(* IEC 61131-3 sources: AXOpen/src/components.siem.identification/ctrl/src/IdentProfile/AxoIdentificationDataTypes, 3 files *)

(* ---- Axo_IID_CMD_STRUCT.st ---- *)
NAMESPACE AXOpen.Components.Siem.Identification
    {S7.extern=ReadWrite}
    CLASS PUBLIC Axo_IID_CMD_STRUCT
        VAR PUBLIC
            CMD			    :   eAxo_IID_COMMANDS;	                    //Command ID
            ATTRIBUTES	    :   BYTE                    :=  BYTE#16#0;	//Subcommands
            OFFSETBUFFER    :   UINT                    :=  UINT#0;     //Offset for receive buffer
            EPCID_UID	    :   ARRAY[1..62] OF BYTE;
            LEN_DATA	    :   WORD                    :=WORD#16#0;	//Length of data
            ADDR_TAG	    :   DWORD                   :=DWORD#16#0;	//physical address on tag
            CONFIG		    :   BYTE                    :=BYTE#16#0;	//Config Mode for Init
            CHAINED		    :   BOOL                    :=FALSE;		//Chained Bit: 1= chained; 0=unchained
            EXT_UHF		    :   Axo_IID_IN_EXT_UHF;	                    //further Atrributes for extended UHF commands
        END_VAR
    END_CLASS
END_NAMESPACE

(* ---- Axo_IID_HW_CONNECT.st ---- *)
NAMESPACE AXOpen.Components.Siem.Identification
(*
+-----------+-------------------------------------------+------------------------------------------------------+---------------------+
|           |             RF61xR/RF68xR                 |                     RF1xxC/RF360R                    |   RF180C/RF170C/MV  |
| Parameter +----------+----------+----------+----------+----------+----------+----------+----------+----------+----------+----------+
|			|   CH01   |   CH02   |   CH03   |   CH04   |   CH01   |   CH02   |   CH03   |   CH04   |CM_CONFIG |   CH01   |   CH02   |
+===========+==========+==========+==========+==========+==========+==========+==========+==========+==========+==========+==========+
| API       | 16#5B00  | 16#5B00  | 16#5B00  | 16#5B00  | 16#5B00  | 16#5B00  | 16#5B00  | 16#5B00  | 16#5B00  |   16#00  |   16#00  |
+-----------+----------+----------+----------+----------+----------+----------+----------+----------+----------+----------+----------+
| SLOT      |     1    |     1    |     1    |     1    |     2    |     3    |     4    |     5    |     1    |     1    |     1    |
+-----------+----------+----------+----------+----------+----------+----------+----------+----------+----------+----------+----------+
| SUB_SLOT  |     1    |     1    |     1    |     1    |     1    |     1    |     1    |     1    |     1    |     1    |     1    |
+-----------+----------+----------+----------+----------+----------+----------+----------+----------+----------+----------+----------+
|CM_CHANNEL |     1    |     2    |     3    |     4    |     1    |     1    |     1    |     1    |     1    |     1    |     2    |
+-----------+----------+----------+----------+----------+----------+----------+----------+----------+----------+----------+----------+
*)
    {S7.extern=ReadWrite}
    CLASS PUBLIC Axo_IID_HW_CONNECT
        VAR PUBLIC
            HW_ID               :   WORD    :=  WORD#16#0; 			//Hardware identifier
            AR_NUMBER 			:   WORD    :=  WORD#16#0; 			//Number of AR
            API 				:   DWORD   :=  DWORD#16#0000_5B00; //API number
            SLOT 				:   WORD    :=  WORD#16#02;  		//Slot number
            SUB_SLOT 			:   WORD    :=  WORD#16#01; 		//Subslot number
            CM_CHANNEL 			:   UINT    :=  UINT#1; 		    //channel of communication module
            Static              :   Axo_IID_IN_SYNC;
        END_VAR
    END_CLASS
END_NAMESPACE

(* ---- AxoByteArray256.st ---- *)
NAMESPACE AXOpen.Components.Siem.Identification
    {S7.extern=ReadWrite}
    CLASS PUBLIC AxoByteArray256 EXTENDS AXOpen.Core.AxoByteArray
        VAR PUBLIC
            Data : ARRAY [0..255] OF BYTE;
        END_VAR
    END_CLASS
END_NAMESPACE
